(* PLC project SafeLOGIC-1, BrAutomation SafeDESIGNER  4.1.3.320 *)
(* stored: companyURL http://www.br-automation.com, creationDateTime Thu May 07 12:54:25 2020 *)

PROGRAM SafeModules_OK

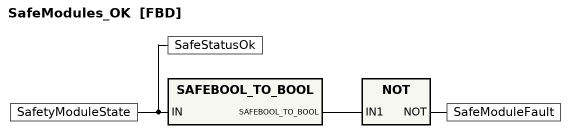
(* FBD diagram, written out as Structured Text *)
SafeStatusOk := SafetyModuleState;
SafeModuleFault := NOT SAFEBOOL_TO_BOOL(SafetyModuleState);
END_PROGRAM
